// TwinCAT 3 PLC project PLC1
// ProgramVersion: 3.1.4024.0
// libraries:
//   Tc2_Standard, * (Beckhoff Automation GmbH)
//   Tc2_System, * (Beckhoff Automation GmbH)
//   Tc3_Module, * (Beckhoff Automation GmbH)
// project tree:
//   DUTs/ Struct_IN.TcDUT, Struct_OUT.TcDUT
//   / PlcTask.TcTTO
//   POUs/ MAIN.TcPOU, Signal_check.TcPOU, Signal_generator.TcPOU
// real-time tasks:
//   TASK PlcTask: cycle T#10ms, priority 20, ADS port 350

CONFIGURATION PLC1
    RESOURCE PLC ON TwinCAT3
        TASK PlcTask(INTERVAL := T#10ms, PRIORITY := 20);
        PROGRAM MAIN WITH PlcTask : MAIN;
    END_RESOURCE
END_CONFIGURATION

// ---- DUTs/Struct_IN.TcDUT
TYPE Struct_IN :
STRUCT
	bHeat2	:	BOOL;
	bOK		:	BOOL;
END_STRUCT
END_TYPE

// ---- DUTs/Struct_OUT.TcDUT
TYPE Struct_OUT :
STRUCT
	bHeat1	:	BOOL;
	bOK		:	BOOL;
	
END_STRUCT
END_TYPE

// ---- POUs/MAIN.TcPOU
PROGRAM MAIN
VAR
	Signal_IN		:	Signal_generator;
	checking		:	Signal_check;
	data_out		:	Struct_OUT;
END_VAR

Signal_IN();
checking(Signal_IN:= Signal_IN.SIGNAL);
data_out.bHeat1 := checking.Signal_OUT;
data_out.bOK := checking.bOK;

END_PROGRAM

// ---- POUs/Signal_generator.TcPOU
FUNCTION_BLOCK Signal_generator
VAR_INPUT
	T		:	TIME	:= T#2S;
END_VAR
VAR_OUTPUT
	SIGNAL	:	BOOL	:= TRUE;
END_VAR
VAR
	timer	:	TON;
END_VAR

timer(IN:= NOT timer.Q, PT:=T/2);
IF timer.Q THEN
	SIGNAL := NOT SIGNAL;
END_IF

END_FUNCTION_BLOCK

// ---- POUs/Signal_check.TcPOU
FUNCTION_BLOCK Signal_check
VAR_INPUT
	Signal_IN	:		BOOL;
	T			:		TIME	:=T#2S;
END_VAR
VAR_OUTPUT
	bOK			:		BOOL	:= TRUE;
	Signal_OUT  :		BOOL;
END_VAR
VAR
	Signal		:		Signal_generator;
	rtrig		:		R_TRIG;
	timer		:		TON;
END_VAR

Signal(T:=T);
Signal_OUT := Signal.SIGNAL;

rtrig(CLK:= Signal_IN);
timer(IN:=  NOT timer.Q, PT:=2*T);		(* rising edge must 
											be detected during 2 periods TO receive bOK := TRUE *)


IF timer.ET < timer.PT THEN
	IF rtrig.Q THEN
		timer.IN:= FALSE;
		bOK := TRUE;
	END_IF
ELSE
	bOK	:= FALSE;
END_IF

END_FUNCTION_BLOCK
